// TIA Portal V18 export
FUNCTION_BLOCK "monitor_perifery"   // FB55, FBD
{ S7_Optimized_Access := 'TRUE' }
VERSION : 0.1
// stored: AutoNumber true, IsIECCheckEnabled false, IsRetainMemResEnabled false, MemoryReserve 100, SetENOAutomatically false, UDAEnableTagReadback false
   VAR_INPUT
      ptDelayed : Time := T#1m;
      inWord : Byte;
      ptMax : Time := T#300ms;
      xBitON : Bool;
   END_VAR
   VAR_OUTPUT
      outWord : Byte;
      yERCOMM : Bool;
      yWNdelay : Bool;
      yAllModulesLive : Bool;
   END_VAR
   VAR
      IEC_Timer_0_Instance { S7_SetPoint := 'True'} : TON_TIME;
      startup { S7_SetPoint := 'True'} : TON_TIME;
      delayPassed : Bool;
   END_VAR
BEGIN

REGION Network 1
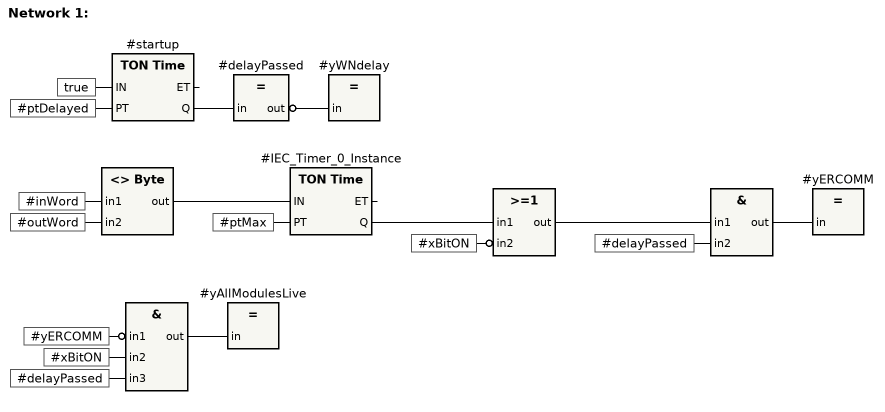
   #startup(IN := true, PT := #ptDelayed);   // TON
   #delayPassed := #startup.Q;
   #yWNdelay := NOT #startup.Q;
   #IEC_Timer_0_Instance(IN := #inWord <> #outWord, PT := #ptMax);   // TON
   #yERCOMM := (#IEC_Timer_0_Instance.Q OR NOT #xBitON) AND #delayPassed;
   #yAllModulesLive := NOT #yERCOMM AND #xBitON AND #delayPassed;
END_REGION

REGION Network 2 (SCL)
   IF (#inWord = #outWord) THEN
       IF #outWord < 100 THEN
           #outWord := #outWord + 1;
       ELSE
           #outWord := 1;
       END_IF;
   END_IF;
END_REGION
END_FUNCTION_BLOCK
